TYPE ST_TONP :
STRUCT
	ET				:TIME;
	Q				:BOOL;
END_STRUCT
END_TYPE

(* stored: Version 1.1.0.1, ProductVersion 3.1.4024.12
   DUT ST_TONP: Id {43e17b6c-4732-4f7f-a629-88d71ccdb24c} *)
